FUNCTION_BLOCK Test_TExecutionWhenBusy_Abort_SelectsAborting EXTENDS T_UnitTestbase
VAR
    Execution : T_Execution;
END_VAR

// Setup...
Execution.FB_init(bInitRetains := FALSE,
                  bInCopyCode  := FALSE);

// Test...
Execution.Start();
Execution.SetBusy();
Execution.Abort();

Assertion.AssertEquals_BOOL(Expected     := TRUE,
                            Actual       := Execution.Aborting,
                            VariableName := 'Execution.Aborting');

TestFinished();

END_FUNCTION_BLOCK

(* stored: Version 1.1.0.1, ProductVersion 3.1.4024.6
   POU Test_TExecutionWhenBusy_Abort_SelectsAborting: Id {62c983db-2c62-4a10-8a80-0b343b0f7d47}, SpecialFunc None *)
